SUBAPPLICATION logiBUS_IXA_TO_CLIENT_OPC (* Digitaler Eingang, aktiver Remote-OPC-UA-Write auf ein ANDERES Geraet via CLIENT_1_0 - 'SUB style': das Protokoll (CLIENT_1_0) steckt IM Baustein selbst, nicht in der Resource des Geraets *)
  (* Standard: 61499-2; Description: Copyright (c) 2026 Meisterschulen am Ostbahnhof This program and the accompanying materials are made available under the terms of the Eclipse Public License 2.0 which is available at https://www.eclipse.org/legal/epl-2.0/ SPDX-License-Identifier: EPL-2.0 *)
  (* Version 1.1, 2026-09-18, Franz Höpfinger, Meisterschulen am Ostbahnhof, logiBUS_IXA.INITO auf logiBUS_IXA.REQ zurueckverdrahtet (Selfloop) - loest nach der Initialisierung sofort einen Service-Request aus, statt auf die erste echte Wertaenderung am Bus zu warten (Fix fuer 'Waiting for handle'-Status direkt nach Boot). *)
  (* Version 1.0, 2026-09-02, Franz Höpfinger, Meisterschulen am Ostbahnhof, initial API and implementation and/or initial documentation *)
  PACKAGE MyLib::sys;
  IMPORT logiBUS::io::DI::logiBUS_DI;
  IMPORT logiBUS::io::DI::logiBUS_DI_S;
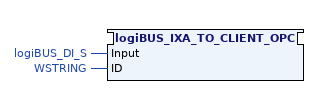
  VAR_INPUT
    Input : logiBUS::io::DI::logiBUS_DI_S := logiBUS_DI::Invalid; (* Identify the Input Input_I1..I8 *)
    ID : WSTRING; (* Remote-Ziel-Adresse (BOOL, ACTION=WRITE, inkl. opc.tcp://-Endpoint des Zielgeraets) *)
  END_VAR
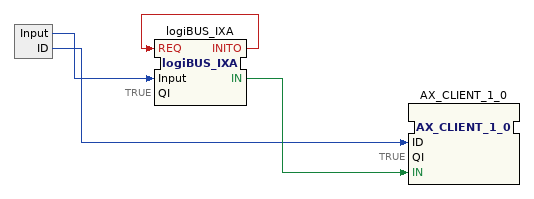
  FBS
    logiBUS_IXA : logiBUS::io::DI::logiBUS_IXA(QI := TRUE);
    AX_CLIENT_1_0 : adapter::net::AX_CLIENT_1_0(QI := TRUE);
  END_FBS
  EVENT_CONNECTIONS
    logiBUS_IXA.INITO TO logiBUS_IXA.REQ;
  END_CONNECTIONS
  DATA_CONNECTIONS
    Input TO logiBUS_IXA.Input;
    ID TO AX_CLIENT_1_0.ID;
  END_CONNECTIONS
  ADAPTER_CONNECTIONS
    logiBUS_IXA.IN TO AX_CLIENT_1_0.IN;
  END_CONNECTIONS
END_SUBAPPLICATION
